FUNCTION_BLOCK FB_Event IMPLEMENTS I_Event
VAR_INPUT
END_VAR
VAR_OUTPUT
END_VAR
VAR
	iHandler:			I_Handler;
	bVerbose:			BOOL;
	bInfo:				BOOL;
	bWarning:			BOOL;
	bError:				BOOL;
	bCritical:			BOOL;	
	stVerbose:			ST_Event;
	stInfo:				ST_Event;
	stWarning:			ST_Event;
	stError:			ST_Event;
	stCritical:			ST_Event;
END_VAR

IF bVerbose THEN
	bVerbose:= FALSE;
ELSE
	stVerbose.nTimestamp:= 0;
END_IF

IF bInfo THEN
	bInfo:= FALSE;	
ELSE
	stInfo.nTimestamp:= 0;		
END_IF

IF bWarning THEN
	bWarning:= FALSE;	
ELSE
	stWarning.nTimestamp:= 0;	
END_IF

IF bError THEN
	bError:= FALSE;	
ELSE
	stError.nTimestamp:= 0;	
END_IF
	
IF bCritical THEN
	bCritical:= FALSE;	
ELSE
	stCritical.nTimestamp:= 0;	
END_IF

METHOD M_Critical
VAR_INPUT
	eType:		E_Type;
	sMessage:	STRING(255);
	nID:		DINT;
END_VAR
bCritical:= TRUE;
IF stCritical.nTimestamp = 0 THEN
	stCritical.nTimestamp:= F_GetSystemTime();
END_IF
stCritical.eEvent:= E_Event.Critical;
stCritical.eType:= eType;
stCritical.sMessage:= sMessage;
stCritical.nID:= nID;

IF iHandler <> 0 THEN
	iHandler.M_Request(stCritical);
END_IF
END_METHOD

METHOD PUBLIC M_Error
VAR_INPUT
	eType:		E_Type;
	sMessage:	STRING(255);
	nID:		DINT;
END_VAR
bError:= TRUE;
IF stError.nTimestamp = 0 THEN
	stError.nTimestamp:= F_GetSystemTime();
END_IF
stError.eEvent:= E_Event.Critical;
stError.eType:= eType;
stError.sMessage:= sMessage;
stError.nID:= nID;

IF iHandler <> 0 THEN
	iHandler.M_Request(stError);
END_IF
END_METHOD

METHOD PUBLIC M_Info
VAR_INPUT
	eType:		E_Type;
	sMessage:	STRING(255);
	nID:		DINT;
END_VAR
bInfo:= TRUE;
IF stInfo.nTimestamp = 0 THEN
	stInfo.nTimestamp:= F_GetSystemTime();
END_IF
stInfo.eEvent:= E_Event.Critical;
stInfo.eType:= eType;
stInfo.sMessage:= sMessage;
stInfo.nID:= nID;

IF iHandler <> 0 THEN
	iHandler.M_Request(stInfo);
END_IF
END_METHOD

METHOD PUBLIC M_Verbose
VAR_INPUT
	eType:		E_Type;
	sMessage:	STRING(255);
	nID:		DINT;
END_VAR
bVerbose:= TRUE;
IF stVerbose.nTimestamp = 0 THEN
	stVerbose.nTimestamp:= F_GetSystemTime();
END_IF
stVerbose.eEvent:= E_Event.Critical;
stVerbose.eType:= eType;
stVerbose.sMessage:= sMessage;
stVerbose.nID:= nID;

IF iHandler <> 0 THEN
	iHandler.M_Request(stVerbose);
END_IF
END_METHOD

METHOD M_Warning
VAR_INPUT
	eType:		E_Type;
	sMessage:	STRING(255);
	nID:		DINT;
END_VAR
bWarning:= TRUE;
IF stWarning.nTimestamp = 0 THEN
	stWarning.nTimestamp:= F_GetSystemTime();
END_IF
stWarning.eEvent:= E_Event.Critical;
stWarning.eType:= eType;
stWarning.sMessage:= sMessage;
stWarning.nID:= nID;

IF iHandler <> 0 THEN
	iHandler.M_Request(stWarning);
END_IF
END_METHOD

PROPERTY PUBLIC P_Handler : I_Handler
GET
P_Handler:= iHandler;
END_GET
SET
iHandler:= P_Handler;
END_SET
END_PROPERTY

END_FUNCTION_BLOCK

(* stored: Version 1.1.0.1, ProductVersion 3.1.4024.12
   POU FB_Event: Id {1dcb84ec-d695-4d6f-a3ff-99e012891880}, SpecialFunc None
   Method M_Critical: Id {43596335-43a4-41c1-ad2f-b3552e29dcfa}
   Method M_Error: Id {5d080c91-569f-424a-821e-4296fce43891}
   Method M_Info: Id {d7d83d14-1059-441b-8e79-b513a6fba4c9}
   Method M_Verbose: Id {51e168c5-af65-4a41-9856-1decc56cb137}
   Method M_Warning: Id {da4a05a4-d352-4379-97c7-69430f6a9b91}
   Property P_Handler: Id {47eda2e3-f16a-4044-b37b-35367509189b}
   Get Get: Id {539e947b-f005-4d1f-9833-5c2b5c69a723}
   Set Set: Id {76fd1b75-9a5b-43f6-8e2f-6b1bcc67aaf5} *)
